// TIA Portal V16 export
// export: Created 2022-02-28T20:45:45.3488768Z, ExportSetting WithDefaults, DisplayName Totally Integrated Automation Portal, DisplayVersion V16, DisplayName TIA Portal Version Control Interface, DisplayVersion V16, DisplayName TIA Portal Openness, DisplayVersion V16, DisplayName STEP 7 Professional, DisplayVersion V16, DisplayName STEP 7 Safety, DisplayVersion V16, DisplayName WinCC Advanced, DisplayVersion V16
FUNCTION "07_Alarmas" : Void   // FC7, LAD
TITLE = Alarmas
{ S7_Optimized_Access := 'TRUE' }
VERSION : 0.1
// stored: AutoNumber true, IsIECCheckEnabled false, SetENOAutomatically false, UDAEnableTagReadback false
BEGIN

REGION Network 1: Paro Emergencia Pistilos
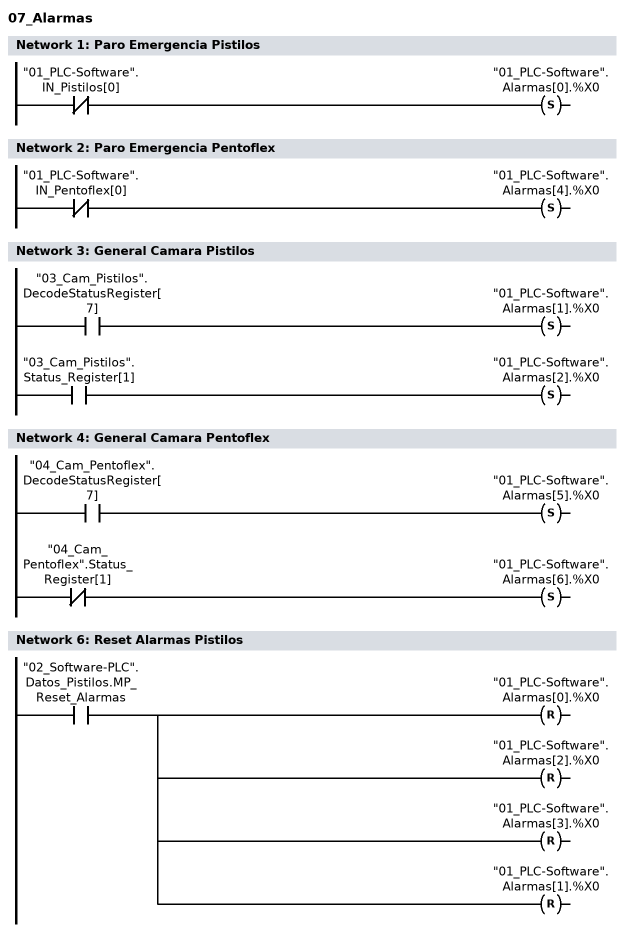
   RUNG wire#powerrail
      I_Contact( "01_PLC-Software".IN_Pistilos[0] )
      S_Coil( "01_PLC-Software".Alarmas[0].%X0 )
   END_RUNG
   // the same network as SCL:
   IF NOT "01_PLC-Software".IN_Pistilos[0] THEN "01_PLC-Software".Alarmas[0].%X0 := TRUE; END_IF;
END_REGION

REGION Network 2: Paro Emergencia Pentoflex
   RUNG wire#powerrail
      I_Contact( "01_PLC-Software".IN_Pentoflex[0] )
      S_Coil( "01_PLC-Software".Alarmas[4].%X0 )
   END_RUNG
   // the same network as SCL:
   IF NOT "01_PLC-Software".IN_Pentoflex[0] THEN "01_PLC-Software".Alarmas[4].%X0 := TRUE; END_IF;
END_REGION

REGION Network 3: General Camara Pistilos
   RUNG wire#powerrail
      Contact( "03_Cam_Pistilos".DecodeStatusRegister[7] )
      S_Coil( "01_PLC-Software".Alarmas[1].%X0 )
   END_RUNG
   RUNG wire#powerrail
      Contact( "03_Cam_Pistilos".Status_Register[1] )
      S_Coil( "01_PLC-Software".Alarmas[2].%X0 )
   END_RUNG
   // the same network as SCL:
   IF "03_Cam_Pistilos".DecodeStatusRegister[7] THEN "01_PLC-Software".Alarmas[1].%X0 := TRUE; END_IF;
   IF "03_Cam_Pistilos".Status_Register[1] THEN "01_PLC-Software".Alarmas[2].%X0 := TRUE; END_IF;
END_REGION

REGION Network 4: General Camara Pentoflex
   RUNG wire#powerrail
      Contact( "04_Cam_Pentoflex".DecodeStatusRegister[7] )
      S_Coil( "01_PLC-Software".Alarmas[5].%X0 )
   END_RUNG
   RUNG wire#powerrail
      I_Contact( "04_Cam_Pentoflex".Status_Register[1] )
      S_Coil( "01_PLC-Software".Alarmas[6].%X0 )
   END_RUNG
   // the same network as SCL:
   IF "04_Cam_Pentoflex".DecodeStatusRegister[7] THEN "01_PLC-Software".Alarmas[5].%X0 := TRUE; END_IF;
   IF NOT "04_Cam_Pentoflex".Status_Register[1] THEN "01_PLC-Software".Alarmas[6].%X0 := TRUE; END_IF;
END_REGION

REGION Network 5: Variador
END_REGION

REGION Network 6: Reset Alarmas Pistilos
   RUNG wire#powerrail
      Contact( "02_Software-PLC".Datos_Pistilos.MP_Reset_Alarmas )
      wire#w1
      R_Coil( "01_PLC-Software".Alarmas[0].%X0 )
   END_RUNG
   RUNG wire#w1
      R_Coil( "01_PLC-Software".Alarmas[2].%X0 )
   END_RUNG
   RUNG wire#w1
      R_Coil( "01_PLC-Software".Alarmas[3].%X0 )
   END_RUNG
   RUNG wire#w1
      R_Coil( "01_PLC-Software".Alarmas[1].%X0 )
   END_RUNG
   // the same network as SCL:
   IF "02_Software-PLC".Datos_Pistilos.MP_Reset_Alarmas THEN
       "01_PLC-Software".Alarmas[0].%X0 := FALSE;
       "01_PLC-Software".Alarmas[2].%X0 := FALSE;
       "01_PLC-Software".Alarmas[3].%X0 := FALSE;
       "01_PLC-Software".Alarmas[1].%X0 := FALSE;
   END_IF;
END_REGION
END_FUNCTION
